Staubli VAL3: OnF5.pgx

program OnF5()
begin

  //

end
